(* IEC 61131-3 sources: programs/VI-54/VI-54_20171205/VI-54_20171205/Stations/PLC_VI54/VI-54_171014/Class/MachineBase, 1 file *)

(* ---- MachineBase.st ---- *)
(*!
<Class
	Name               = "MachineBase"
	Revision           = "0.0"
	RealtimeTask       = "false"
	CyclicTask         = "false"
	BackgroundTask     = "false"
	Sigmatek           = "false"
	OSInterface        = "false"
	HighPriority       = "false"
	Automatic          = "false"
	UpdateMode         = "Prescan"
	SharedCommandTable = "true"
	Objectsize         = "(600,240)">
	<Channels>
		<Server Name="ObjectServer" Visualized="false" Initialize="false" WriteProtected="false" Retentive="false"/>
		<Server Name="RunningMode" Visualized="true" Initialize="false" WriteProtected="true" Retentive="false"/>
		<Server Name="Stepper" Visualized="true" Initialize="false" WriteProtected="false" Retentive="false"/>
		<Client Name="Standaard" Required="true" Internal="true"/>
	</Channels>
	<Network Name="MachineBase">
		<!-- List of Components in this network -->
		<Components>
			<Object
				Name       = "Standaard"
				Class      = "Standard"
				Position   = "(120,210)"
				Visualized = "false">
				<Channels>
					<Server Name="ClassSvr"/>
				</Channels>
			</Object>
		</Components>
		<Comments>
		</Comments>
		<!-- List of Connections in this network -->
		<Connections>
			<Connection Source="this.Standaard" Destination="Standaard.ClassSvr"/>
		</Connections>
		<!-- Headerfiles -->
		<Options>
		</Options>
	</Network>
</Class>
*)
MachineBase : CLASS
  //Servers:
	ObjectServer 	: SvrChCmd_DINT;
	Stepper 	: SvrCh_DINT;
	RunningMode 	: SvrCh_RunningStateEnum;
  //Clients:
	Standaard 	: CltChCmd_Standard;
  //Variables:
		GlobalDataPtr 	: ^GlobalDataStr;
		RecipePtr 	: ^DataRecipeStr;
  //Functions:

	FUNCTION VIRTUAL GLOBAL MyInit;

	FUNCTION VIRTUAL GLOBAL MyRtTask;

	FUNCTION VIRTUAL GLOBAL MyCyTask;

	FUNCTION VIRTUAL GLOBAL MyBackTask;

	FUNCTION GLOBAL SetGlobalDataPtr
		VAR_INPUT
			Ptr 	: ^GlobalDataStr;
		END_VAR
		VAR_OUTPUT
			ReturnPtr 	: ^GlobalDataStr;
		END_VAR;

	FUNCTION GLOBAL RtTask;

	FUNCTION GLOBAL CyTask;

	FUNCTION GLOBAL BgTask;

	FUNCTION GLOBAL InitTask
		VAR_INPUT
			SetGlobalPtr 	: ^GlobalDataStr;
			SetRecipePtr 	: ^DataRecipeStr;
		END_VAR;

	FUNCTION VIRTUAL GLOBAL ResetErrors;
  //Tables:
	FUNCTION @STD
		VAR_OUTPUT
			ret_code	: CONFSTATES;
		END_VAR;
	FUNCTION GLOBAL TAB @CT_;
END_CLASS;

#pragma using Standard

FUNCTION VIRTUAL GLOBAL MachineBase::MyInit

    // alleen bij firstscan

END_FUNCTION

FUNCTION VIRTUAL GLOBAL MachineBase::MyRtTask

    // Real time task

END_FUNCTION

FUNCTION VIRTUAL GLOBAL MachineBase::MyCyTask

    //  Cycle time task

END_FUNCTION

FUNCTION VIRTUAL GLOBAL MachineBase::MyBackTask

    // Background task

END_FUNCTION

FUNCTION GLOBAL MachineBase::SetGlobalDataPtr
	VAR_INPUT
		Ptr 	: ^GlobalDataStr;
	END_VAR
	VAR_OUTPUT
		ReturnPtr 	: ^GlobalDataStr;
	END_VAR

  GlobalDataPtr := Ptr;

  ReturnPtr := GlobalDataPtr;

END_FUNCTION

FUNCTION GLOBAL MachineBase::RtTask

  MyRtTask();

END_FUNCTION

FUNCTION GLOBAL MachineBase::CyTask

  RunningMode := GlobalDataPtr^.gRunStatus.gRunStatusGlob;
  MyCyTask();

END_FUNCTION

FUNCTION GLOBAL MachineBase::BgTask

  Standaard.Background(EAX := 0);
  MyBackTask();

END_FUNCTION

FUNCTION GLOBAL MachineBase::InitTask
	VAR_INPUT
		SetGlobalPtr 	: ^GlobalDataStr;
		SetRecipePtr 	: ^DataRecipeStr;
	END_VAR

  // alleen bij firstscan
  GlobalDataPtr := SetGlobalPtr;
  RecipePtr     := SetRecipePtr;

  MyInit();

END_FUNCTION

FUNCTION VIRTUAL GLOBAL MachineBase::ResetErrors

END_FUNCTION
